# EPICS autosave request: ADApp/Db/ADAsyn_settings.req
$(P)$(D)BinX
$(P)$(D)BinY
$(P)$(D)FilePath
$(P)$(D)FileName
$(P)$(D)FileNumber
$(P)$(D)AutoIncrement
$(P)$(D)FileTemplate
$(P)$(D)AutoSave
